FUNCTION F_SetZoneOccupiedEmulation : BOOL
(**************************************************************************************
 * 	Application		:	BoxControl Framework
 *	Revision		:	$Revision: 404529 $
 *	Revision date	:	$Date: 2018-04-23 08:21:38 +0200 (Mo., 23 Apr 2018) $
 *	Last changed by	:	$Author: b7bolm $
 *	URL				:	$URL: http://almscdc.swisslog.com/repo/SWPD/Development/BoxControlFramework/20_Release/trunk/01_Software/BCF/BCF/JumpStart/20_Product/11_Emu/12_E_Functions/10_Lib/10_Conv/10_Functions/F_SetZoneOccupiedEmulation.TcPOU $
 *
 *	Purpose			:	Set HW input zone occupied 
 *
 * ------------------------------------------------------------------------------------
 *	Copyright Swisslog [IP AG], Switzerland. All rights reserved.
 * 
 * ------------------------------------------------------------------------------------
 *	
 * 	Revision History: 
 *
 * 	VERSION			DATE			INITIALS			DESCRIPTION
 *	0.1				01.01.2001		swl					Example
 *
 **************************************************************************************)
VAR_INPUT
	eFunctionNumber	: E_FunctionNumber; // Function number
	ZoneNumber		: INT; // Zone number
	Occupied  		: BOOL; // Occupied state
END_VAR
VAR
	SetHW_Input 	: ST_SetHW_Inputs;
	EnableHW_Input  : ST_SetHW_Inputs;
END_VAR

// Check if function number is valid
IF eFunctionNumber > E_FunctionNumber.F_BEGIN_FUNCTION AND
   eFunctionNumber < E_FunctionNumber.F_END_FUNCTION THEN

	// Check reference is valid
	IF __ISVALIDREF(FunctionRegistryEmulation[eFunctionNumber].rFunction) THEN
   		// Process HW inputs
		SetHW_Input.Occupied[1] 	:= Occupied;
		EnableHW_Input.Occupied[1] 	:= TRUE;
		FunctionRegistryEmulation[eFunctionNumber].rFunction.M_SetHW_Inputs(mZoneNumber:= ZoneNumber, mSetHW_Input:= SetHW_Input, mEnableHW_Input:= EnableHW_Input);
	END_IF
END_IF

END_FUNCTION

(* stored: Version 1.1.0.1, ProductVersion 3.1.4022.12
   POU F_SetZoneOccupiedEmulation: Id {19dc2591-fa38-4b74-9557-a67e3e0f2966}, SpecialFunc None *)
